{attribute wpf [Container(Layout.Stack)]}
FUNCTION_BLOCK NotificationPanel EXTENDS TcoObject
VAR_INPUT
	(*~
		<docu>
			<summary>
				Time duration for toggle signal.
			</summary>
		</docu>
	~*)
	inBlinkPeriod:TIME;
END_VAR

VAR
	{attribute addProperty Name "<#Heart beat#>"}
  	_heartBeat : BOOL;
	
    {attribute clr [RenderIgnore()]}
	_badgeValue : INT;

	{attribute clr [RenderIgnore()]}
    _toggle: TcoUtilities.TcoBlinker(THIS^);
	
	_iconSet: ARRAY[0..20] OF Icon; //ak potrebujes zobrazit viac ikon, uprav velkost pola
	
	_iconSetClear : ARRAY[0..20] OF Icon; //ak potrebujes zobrazit viac ikon, uprav velkost pola
	
	_iconPlcPulse : Icon;
	
	_iconParamsClear : Icon;
	
END_VAR



_iconPlcPulse.Title := '<#PLC connection#>';
_iconPlcPulse.IconType := TO_STRING(eIconType.plcConnection);
_iconPlcPulse.Signal := _heartBeat;
_iconPlcPulse.DisableRedIcon := TRUE;
addIcon(_iconPlcPulse);

//setIconsStyle();

Blink();
CountSignals();

METHOD AddIcon : BOOL
VAR_INPUT
	inIcon : Icon;
END_VAR

VAR 
	_index : INT;
END_VAR
FOR  _index := 0 TO 20 DO 
	IF _IconSet[_index].Title = '' THEN
		_IconSet[_index] := inIcon;
		RETURN;
	END_IF
END_FOR
END_METHOD

METHOD Blink
VAR 
	_index : INT;
END_VAR
_toggle(inOffTime:=inBlinkPeriod,inOnTime:=inBlinkPeriod);
_heartBeat := _toggle.IsOn;
	FOR _index := 0 TO 20 DO
		IF _iconSet[_index].BlinkEnabled AND NOT _iconSet[_index].Signal THEN 
			_iconSet[_index].SignalBlink := _toggle.IsOn;		
		ELSE
			_iconSet[_index].SignalBlink := _iconSet[_index].Signal;
		END_IF
	END_FOR
END_METHOD

METHOD Clear
_iconSet := _iconSetClear;
_badgeValue := 0;
END_METHOD

METHOD CountSignals
VAR
	_iconIndex : INT;
END_VAR
_iconIndex := 0;
_badgeValue := 0;
FOR _iconIndex := 0 TO 20 DO
	IF _iconSet[_iconIndex].Title <> '' AND  NOT _iconSet[_iconIndex].DisableRedIcon THEN 
		_badgeValue := _badgeValue + BOOL_TO_INT(NOT _iconSet[_iconIndex].Signal);
	END_IF
END_FOR
END_METHOD

METHOD PRIVATE setIconsStyle
VAR 
	_index : INT;
END_VAR
//FOR _index := 0 TO 20 DO 
//	CASE _iconSet[_index].IconType OF 
//		eIconType.controlVoltage : _iconSet[_index].IconType := 'Power';
//		eIconType.airPressure : _iconSet[_index].IconType := 'OxygenTank';
//		eIconType.emergencyStop : _iconSet[_index].IconType := 'Alert';
//		eIconType.safetyDoor : _iconSet[_index].IconType := 'ShieldCheck';
//		eIconType.doorClosed : _iconSet[_index].IconType := 'Door';
//		eIconType.doorLocked : _iconSet[_index].IconType := 'DoorClosedLock';
//		eIconType.processDataLoaded : _iconSet[_index].IconType := 'CogOutline';
//		eIconType.technologyDataLoaded : _iconSet[_index].IconType := 'ClipboardCheckOutline';
//		eIconType.opticBarrier : _iconSet[_index].IconType := 'Hand';
//		eIconType.robot : _iconSet[_index].IconType := 'RobotIndustrial';
//		eIconType.plcConnection : _iconSet[_index].IconType := 'HeartPulse';
//	ELSE
//		 _iconSet[_index].IconType := _iconSet[_index].IconType;
//	END_CASE
//END_FOR
END_METHOD

METHOD SetSignal
VAR_INPUT
	inTitle : STRING;
	inSignal : BOOL;
END_VAR

VAR
	_index : INT;
END_VAR
FOR _index := 0 TO 20 DO 
	IF _iconSet[_index].Title = inTitle THEN 
		_iconSet[_index].Signal := inSignal;
		RETURN;
	END_IF
END_FOR
END_METHOD

END_FUNCTION_BLOCK

(* stored: Version 1.1.0.1
   POU NotificationPanel: Id {2928ab2f-ea83-0435-171c-b9c0980f8160}, SpecialFunc None
   Method AddIcon: Id {2a610e16-906a-49b5-9c35-0302376f96c9}
   Method Blink: Id {d779bc9b-5ccc-4241-baac-18a7b45cc3d3}
   Method Clear: Id {98437acd-3427-45b1-8068-68a3fcbfcb6c}
   Method CountSignals: Id {cb041011-57e9-48eb-8354-3b0ea9b4ed06}
   Method setIconsStyle: Id {c2462871-419f-4d9d-b904-af8fc3f6ed34}
   Method SetSignal: Id {665d5821-5d96-4799-aa5d-f419e69d82b5} *)
